VAR_GLOBAL
	rStatus		: REAL;
	bBlink		: BOOL;
END_VAR

(* stored: Version 1.1.0.1
   GVL GVL_Blinker: Id {c0ef48c9-f3ad-44f1-87d2-ce61b64192a3} *)
